/// Read-only interface exposing all output variables of FB_Mfr_WeatherNow (including base class fields).
INTERFACE I_Mfr_WeatherNow

/// Cloud coverage [%].
PROPERTY CloudCoverage : REAL
GET
END_GET
END_PROPERTY

/// Relative humidity [%].
PROPERTY Humidity : REAL
GET
END_GET
END_PROPERTY

/// Precipitation [mm].
PROPERTY Precipitation : REAL
GET
END_GET
END_PROPERTY

/// Atmospheric pressure [hPa].
PROPERTY Pressure : REAL
GET
END_GET
END_PROPERTY

/// Temperature [°C].
PROPERTY Temperature : REAL
GET
END_GET
END_PROPERTY

/// TRUE when the gateway has written valid weather data.
PROPERTY Valid : BOOL
GET
END_GET
END_PROPERTY

/// Visibility [km].
PROPERTY Visibility : REAL
GET
END_GET
END_PROPERTY

/// Weather condition code.
PROPERTY WeatherCondition : E_Mfr_WthCond
GET
END_GET
END_PROPERTY

/// Wind bearing (16 cardinal directions).
PROPERTY WindBearing : E_Mfr_WndBrng
GET
END_GET
END_PROPERTY

/// Wind speed [km/h].
PROPERTY WindSpeed : REAL
GET
END_GET
END_PROPERTY

END_INTERFACE

(* stored: Version 1.1.0.1
   Itf I_Mfr_WeatherNow: Id {e0696dc1-f20d-4aab-a8e4-0627bcaac867}
   Property CloudCoverage: Id {b8b47fdb-30c5-4bba-88d2-06a8059bbb4c}
   Get Get: Id {9fc6892c-642a-48f8-88ed-8b5d4891079c}
   Property Humidity: Id {447e5d52-dacb-43aa-a503-ed1532601fe5}
   Get Get: Id {99456f23-0d27-4c81-8b66-84ca90578e89}
   Property Precipitation: Id {f5274c23-3d23-432b-a230-8bf76971aaa1}
   Get Get: Id {c54c5170-82b0-4b3e-ac2c-ccb7cc583afd}
   Property Pressure: Id {73e212cd-8dc4-4933-9272-a8408324c15f}
   Get Get: Id {04bf96b8-7883-44cc-973e-9ce295413a27}
   Property Temperature: Id {5c85afce-534d-4623-8d6c-7124321aa610}
   Get Get: Id {652f6492-b516-4686-a962-d62fc657f334}
   Property Valid: Id {728340b5-779f-45ca-805f-8cdb69a4530c}
   Get Get: Id {4d5b906e-ad8f-47bf-b32b-bb9f1f9df30e}
   Property Visibility: Id {7e084291-79d3-4060-9b8f-85b05064ad81}
   Get Get: Id {d6fd85cf-afc7-49cb-a67b-40bd91236134}
   Property WeatherCondition: Id {61decf1a-648b-481b-9b7e-3e1bd536d3af}
   Get Get: Id {a0716ca0-44ea-478f-a083-520e5974d116}
   Property WindBearing: Id {2f626eac-ea47-4abc-84a6-081d954c5043}
   Get Get: Id {f33bbc59-c9c1-4318-a769-d4519c79e445}
   Property WindSpeed: Id {6829221d-b2fb-4db4-9aaa-9da65796c977}
   Get Get: Id {f745036f-586d-4ffe-9740-d018b924c03b} *)
